PROGRAM P_AutoMode_Old_Broadcast
VAR
END_VAR

//if it is a night
IF F_IsNight() THEN
	//turn all lights full ON
	GVL_StreetLamps.nDimmValue_B := 255;
ELSE //it is a day
	//turn all lights OFF
	GVL_StreetLamps.nDimmValue_B := 0;
END_IF

END_PROGRAM

(* stored: Version 1.1.0.1, ProductVersion 3.1.4024.5
   POU P_AutoMode_Old_Broadcast: Id {ab93a4bf-d261-45ea-bbfd-2dbe71e42783}, SpecialFunc None *)
